FUNCTION_BLOCK fbUnderPresureTester_V3 IMPLEMENTS I_StationMachine
VAR_IN_OUT
	stInOuts 					: stUnderPressureTesterInOuts_V3;	//In Outs for modules
	stParams					: stUnderPressureTestParams_V3;		//Parameters for underpressure chamber
END_VAR
VAR_INPUT
END_VAR
VAR_OUTPUT
END_VAR
VAR
	fbVacuumMeasure				: 	fbAnalogMeasurement;		//Block for underpressure calibration
	fbTON_1Hz					: 	TON;						//Timer with 1 Hz cycle
	bOneHzClock					: 	BOOL;						//Bool variable for 1 Hz status
	iWorkStep					: 	INT;						//Step in sequence of work
	fbTON_VacumObtained			: 	TON;						//Filtering the vacuum status
	fbTON_VacumNearZero			: 	TON;						//Filtering the vacuum status
	I_PimSystem					: 	I_PIM;						//PIM block
	fbTON_VacuumMonitor			: 	TON;						//Checking that undeerpressure in increasing;			
	rLastUnderPressure			: 	REAL;						//Underpressure history		
	fbTOFF_CycleEndTurnOf		: 	TOF;						//Setting up end cycle
	//iCyclesToRepeat				: 	INT;						//How many cycles need to be done?		
	bServiceReset				: BOOL;							//Reset 
	bManual						: BOOL;							//Manual mode
	fbWorkTimer					: TON;							//Timer for purpose of error
END_VAR

ACT_Background();
CASE iWorkStep OF
	0:		// Init
		iWorkStep := 1;
		stInOuts.bPumpRly := FALSE;
		stInOuts.bEValve := TRUE;
		I_PimSystem.mSetNewMachineState(nPIM_MachineStates._0_Initialization);
	1:		// Wait for obtaining atmospheric pressure
		IF NOT stInOuts.bEValve THEN
			iWorkStep := 5;
		END_IF
	5:		// Setup new test
		I_PimSystem.mSetNewMachineState(nPIM_MachineStates._0_Standby_NotReady);
		iWorkStep := 10;
	10:		// Waiting for ext test premission 
		I_PimSystem.mSetNewMachineState(nPIM_MachineStates._2_ReadyForNewOperation);
		IF stInOuts.bLockSens AND stInOuts.bSafetyOK AND NOT stInOuts.bEValve THEN
			IF I_PimSystem.mSetNewMachineState(nPIM_MachineStates._3_NewOperationStarted) THEN
				iWorkStep := 15;
			END_IF
		END_IF
	15:		// Stating new cycle
		stInOuts.bPumpRly := TRUE;
		I_PimSystem.mSetNewMachineState(nPIM_MachineStates._4_OperationInProgress);
		iWorkStep := 20;
	20:		// Waiting for end of cycle
		IF fbTON_VacumObtained.Q THEN
			stInOuts.bPumpRly := FALSE;
			stInOuts.bEValve := TRUE;
			iWorkStep := 25;
		END_IF
	25:		//Waiting for pressure low value
		IF NOT stInOuts.bEValve THEN
			iWorkStep := 30;
		END_IF
	30:		//Waiting for doors open
		IF NOT stInOuts.bLockSens THEN
			iWorkStep := 5;
		END_IF
	90:	//Error obtained
		I_PimSystem.mSetNewMachineState(nPIM_MachineStates._8_WaitForReset);
		iWorkStep	:= 91;
		stInOuts.bEValve	:= TRUE;
		stInOuts.bPumpRly	:= FALSE;
	91:	//Waiting for reset
		IF I_PimSystem.mSetNewMachineState(nPIM_MachineStates._9_ResetInProgress) OR bServiceReset THEN
			IF stInOuts.bSafetyOK THEN
				stInOuts.bEValve	:= TRUE;
				stInOuts.bPumpRly	:= FALSE;
				iWorkStep			:= 95;
			ELSE
				iWorkStep	:= 90;
			END_IF
		END_IF
	95:	//Reset confirmed
		I_PimSystem.mSetNewMachineState(nPIM_MachineStates._0_Standby_NotReady);
		iWorkStep		:= 5;
END_CASE

ACTION ACT_Background:
//------------------------------------------------------------------------------------------------
//Measurement scalling
fbVacuumMeasure(rIn:=stInOuts.iVacuumLevel,
				stMeasureScalingData:=stParams.stVacuumData,
				tStalaczasowa:= T#10MS,
				rOutFiltered=>stInOuts.rVacuumLevel);
//------------------------------------------------------------------------------------------------
//1Hz clock
fbTON_1Hz(IN:=NOT fbTON_1Hz.Q,PT:=T#500MS);
bOneHzClock := fbTON_1Hz.Q XOR bOneHzClock;
//------------------------------------------------------------------------------------------------
//LED Light Control
stInOuts.bLEDGreen		:= tCycleEnd;
stInOuts.bLEDRed 		:= (NOT stInOuts.bSafetyOK AND bOneHzClock) OR tInErrorState;
stInOuts.bLEDYellow 	:= (iWorkStep = 10) OR (tChamberBusy AND bOneHzClock) ;
stInOuts.bLEDReset 		:= NOT stInOuts.bSafetyOK;
//------------------------------------------------------------------------------------------------
//Vacuum obtained
fbTON_VacumObtained(IN:=stInOuts.rVacuumLevel>=stParams.rVaccumLevelToObtain,PT:=T#50MS);
//------------------------------------------------------------------------------------------------
//No Vacuum - Stable - Turn off 
fbTON_VacumNearZero(IN:=(stInOuts.rVacuumLevel<4), PT:= T#500MS);
stInOuts.bEValve R= fbTON_VacumNearZero.Q;
//------------------------------------------------------------------------------------------------
//Checking increase of underpressure - Error
fbTON_VacuumMonitor(IN:=tChamberBusy AND (stInOuts.rVacuumLevel > rLastUnderPressure), PT:=T#5S);
//------------------------------------------------------------------------------------------------
//Calculating underpressure increasing
IF stInOuts.rVacuumLevel > rLastUnderPressure AND tChamberBusy THEN
	rLastUnderPressure := stInOuts.rVacuumLevel;
ELSIF NOT tChamberBusy THEN
	rLastUnderPressure := 0;
END_IF
//------------------------------------------------------------------------------------------------
// Cycle end status
fbTOFF_CycleEndTurnOf(IN:=fbTON_VacumObtained.Q,PT:=T#5S);
//------------------------------------------------------------------------------------------------
// Error pressure is no increasing 
IF fbTON_VacuumMonitor.Q AND NOT tInErrorState THEN
	mNewEvent(nEventClass:=nPIM_EventClasses.Error,nEvent:=nUnderPressureTestErrorCodes_V3._860_TestTimeOut);
END_IF
//------------------------------------------------------------------------------------------------
//Error safety turned on
IF NOT  stInOuts.bSafetyOK AND NOT tInErrorState THEN
	mNewEvent(nEventClass:=nPIM_EventClasses.Error,nEvent:=nUnderPressureTestErrorCodes_V3._861_SafetyError);
END_IF
//------------------------------------------------------------------------------------------------
// Timer for error
fbWorkTimer(IN:=tChamberBusy,PT:=T#30S);
IF fbWorkTimer.Q THEN
	mNewEvent(nEventClass:=nPIM_EventClasses.Error,nEvent:=nUnderPressureTestErrorCodes_V3._860_TestTimeOut);
END_IF
IF tChamberBusy AND stInOuts.bEValve THEN
	mNewEvent(nEventClass:=nPIM_EventClasses.Error,nEvent:=nUnderPressureTestErrorCodes_V3._864_EjectionValveOpenedDuringTest);
END_IF
END_ACTION

METHOD FB_init : BOOL
VAR_INPUT
	bInitRetains	: BOOL;
	bInCopyCode 	: BOOL;
	I_Pim			: I_PIM;
END_VAR
I_PimSystem := I_Pim;
END_METHOD

{warning 'add method implementation '}
(* Metoda TRUE kiedy dane wyjściowe są ok, jeśli nie FALSE (jeśli not bBusy i FALSE to błąd odczytu) *)
METHOD mGetParamsData : BOOL
VAR_INPUT
	(* Jeśli TRUE metoda okresla czy ma dostęp do parametrów, jeśli tak zwraca TRUE, jeśli nie FALSE*)
	bTestParams	: BOOL;
END_VAR
VAR_OUTPUT
	(* Maszyna odświeża dane*)
	bBusy	: BOOL;
	(* Wskaźnik do parametrów pracy maszyny*)
	pMachineParametersStruct	: POINTER TO BYTE;
	(* Rozmiar struktury parametrów pracy maszyny [bajty]*)
	uiMachineParametersSize	: UINT;
	(* Aktualna suma CRC16 obliczona z parametrów*)
	wActualCRC16SumInMachine	: WORD;
END_VAR
IF bTestParams THEN
	//mGetParamsData := stMachineSettings.bSerialCommunicationEN;
ELSE
	//pMachineParametersStruct := ADR(stParamAktProgramu);
	//uiMachineParametersSize := SIZEOF(stParamAktProgramu);
	wActualCRC16SumInMachine := F_DATA_TO_CRC16_CCITT(pData := pMachineParametersStruct, cbData := uiMachineParametersSize, crc := 16#0000);
	bBusy := FALSE;
	mGetParamsData := TRUE;	
END_IF
END_METHOD

METHOD INTERNAL mNewEvent : BOOL
VAR_INPUT
	nEventClass:nPIM_EventClasses;
	nEvent: nUnderPressureTestErrorCodes_V3;
END_VAR
IF nEventClass = nPIM_EventClasses.AlarmAutoConfirm OR nEventClass = nPIM_EventClasses.Message THEN		// Alarm nieblokadowy
	I_PimSystem.mSetNewMachineState(nPIM_MachineStates._0_Initialization);
	iWorkStep := 90;
ELSE
	I_PimSystem.mSetNewMachineState(nPIM_MachineStates._7_ErrorOccurr);

	I_PimSystem.mNewEvent(iEventId := nEvent, nEventType := nEventClass, tMessageTime := T#0S);
	iWorkStep := 90;
END_IF
END_METHOD

TRANSITION tChamberBusy:
tChamberBusy := stInOuts.bPumpRly;;
END_TRANSITION

TRANSITION tCycleEnd:
tCycleEnd := fbTOFF_CycleEndTurnOf.Q;
END_TRANSITION

TRANSITION tInErrorState:
tInErrorState := iWorkStep >= 90;
END_TRANSITION

END_FUNCTION_BLOCK

(* stored: Version 1.1.0.1, ProductVersion 3.1.4024.13
   POU fbUnderPresureTester_V3: Id {ec9c1291-17a5-4534-9760-1d0ca5382d72}, SpecialFunc None
   Action ACT_Background: Id {caa100ef-1062-4ed3-a746-3cabb0fe0e32}
   Method FB_init: Id {5f7c60d6-e86b-4311-b062-eaa71e0895c4}
   Method mGetParamsData: Id {5ee79e83-373b-49bb-bdd4-d228e97b9bda}
   Method mNewEvent: Id {3c17e6dc-86ff-404f-824e-72f48088c2bf}
   Transition tChamberBusy: Id {d9c0de54-cfb5-49af-b793-4cc3cc7902a0}
   Transition tCycleEnd: Id {4940a4ee-0e0e-4194-86bc-2521ceb923ae}
   Transition tInErrorState: Id {0d90573e-81c5-45df-af52-9de005e2bd00} *)
